// TIA Portal V19 export
TYPE "LEXCHANGETRAY_typeSR1000ControlNode"
// commands: LEXCHANGETRAY_typeSR1000ControlNodeCommands
// monitoring: LEXCHANGETRAY_typeSR1000ControlNodeMonitoring
// stored: Access Published
   STRUCT
      commands { S7_SetPoint := 'True'} : "LEXCHANGETRAY_typeSR1000ControlNodeCommands";
      monitoring { S7_SetPoint := 'True'} : "LEXCHANGETRAY_typeSR1000ControlNodeMonitoring";
   END_STRUCT;
END_TYPE
